// TIA Portal project "IOT2050_S7_CompleteProject" (V16)

(* hardware
DEVICE "ET 200SP station_1"  ET 200SP-Station
   slot 0: "Rack_0"  Rack  6ES5 710-8MAx1
   slot 1: "PLC_1"  CPU 1512SP F-1 PN  6ES7 512-1SK01-0AB0  V2.5
   slot 2: "Server module_1"  Server module  6ES7 193-6PA00-0AA0  V1.1
      slot 1: "Server module_1"  Server module
   slot 127: "BA 2xRJ45"  BA 2xRJ45  6ES7 193-6AR00-0AA0  V0.0
      slot 32769: "Port_1"  6ES7 193-6AR00-0AA0
      slot 32770: "Port_2"  6ES7 193-6AR00-0AA0
*)

// ===== PLC "PLC_1"  CPU 1512SP F-1 PN =====

DATA_BLOCK "motorControl_DB"   // DB2
{ S7_Optimized_Access := 'TRUE' }
VERSION : 0.1
// stored: InstanceOfName motorControl
"motorControl"
BEGIN
END_DATA_BLOCK

// folder: 01_S7

DATA_BLOCK "S7_Data"   // DB1
{ S7_Optimized_Access := 'FALSE' }
VERSION : 0.1
   VAR
      TO_IOT2050 : Struct
         motorCurrent : UInt;   // measured in Amps. Value range (0-255)
         motorVoltage : UInt;   // measured in Volts. Value range (0-255)
         motorTemperature : Real;   // measured in °C
         motorStatus : Bool;   // 0: motor off; 1: motor running (on)
      END_STRUCT;
      FROM_IOT2050 : Struct
         controlButton : Bool;   // button to start or stop motor
      END_STRUCT;
   END_VAR
BEGIN
END_DATA_BLOCK

// folder: (top level)

ORGANIZATION_BLOCK "Main"   // OB1, LAD, ProgramCycle
TITLE = "Main Program Sweep (Cycle)"
{ S7_Optimized_Access := 'TRUE' }
VERSION : 0.1
   VAR_INPUT
      Initial_Call : Bool;   // Initial call of this OB
      Remanence : Bool;   // =True, if remanent data are available
   END_VAR
BEGIN

REGION Network 1
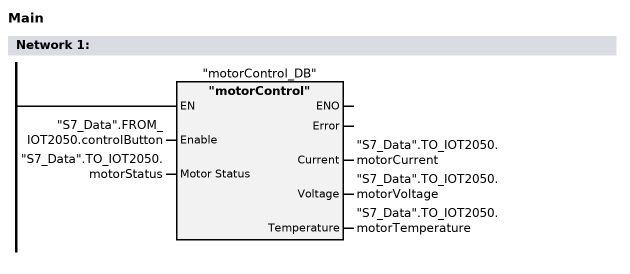
   RUNG wire#powerrail
      "motorControl_DB"(Enable := "S7_Data".FROM_IOT2050.controlButton, "Motor Status" := "S7_Data".TO_IOT2050.motorStatus, Error =>, Current => "S7_Data".TO_IOT2050.motorCurrent, Voltage => "S7_Data".TO_IOT2050.motorVoltage, Temperature => "S7_Data".TO_IOT2050.motorTemperature)
   END_RUNG
   // the same network as SCL:
   "motorControl_DB"(Enable := "S7_Data".FROM_IOT2050.controlButton,   // "motorControl"
                     "Motor Status" := "S7_Data".TO_IOT2050.motorStatus,
                     Current => "S7_Data".TO_IOT2050.motorCurrent,
                     Voltage => "S7_Data".TO_IOT2050.motorVoltage,
                     Temperature => "S7_Data".TO_IOT2050.motorTemperature);
END_REGION
END_ORGANIZATION_BLOCK

// folder: 01_S7

FUNCTION_BLOCK "motorControl"   // FB1, LAD
{ S7_Optimized_Access := 'TRUE' }
VERSION : 0.1
   VAR_INPUT
      Enable : Bool;
   END_VAR
   VAR_OUTPUT
      Error : Bool;
      Current : UInt;
      Voltage : UInt;
      Temperature : Real;
   END_VAR
   VAR_IN_OUT
      "Motor Status" : Bool;
   END_VAR
   VAR
      LGF_SinusCI_Instance : "LGF_SinusCI";
      LGF_RectangleCI_Instance : "LGF_RectangleCI";
   END_VAR
   VAR_TEMP
      randIntError : Bool;
      randIntStatusID : UInt;
      randIntStatus : Word;
      sinusError : Bool;
      sinusStatusID : UInt;
      sinusStatus : Word;
      rectError : Bool;
      rectStatusID : UInt;
      rectStatus : Word;
   END_VAR
BEGIN

REGION Network 1: Set the Motor status to ON/OFF and turn ON/OFF the motor
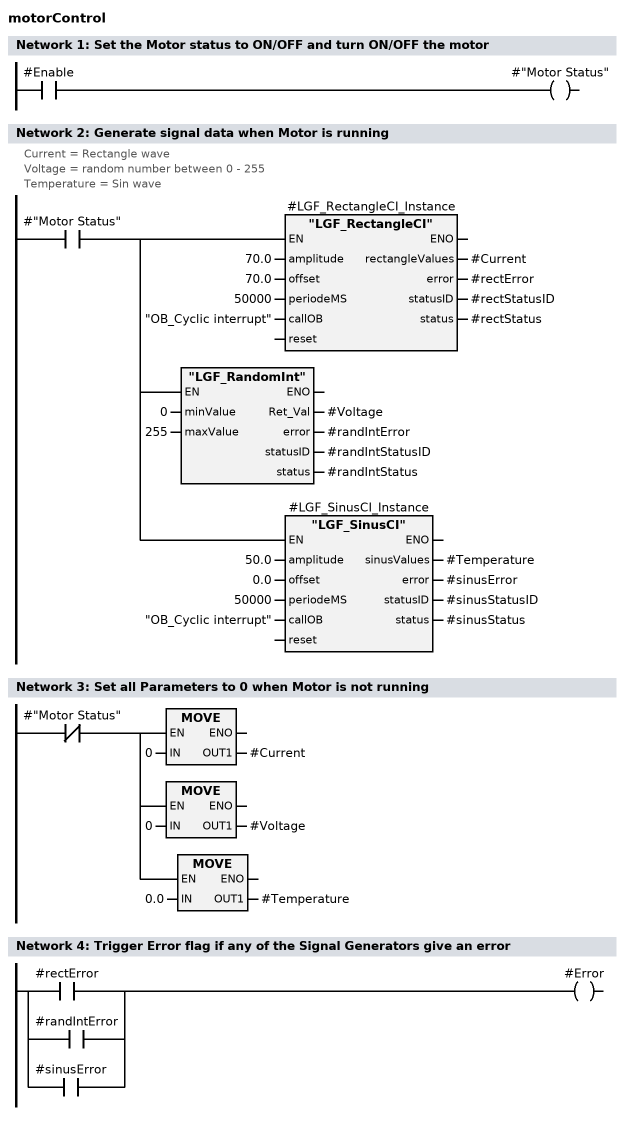
   RUNG wire#powerrail
      Contact( #Enable )
      Coil( #"Motor Status" )
   END_RUNG
   // the same network as SCL:
   #"Motor Status" := #Enable;
END_REGION

REGION Network 2: Generate signal data when Motor is running
   // Current = Rectangle wave
   // Voltage = random number between 0 - 255
   // Temperature = Sin wave
   RUNG wire#powerrail
      Contact( #"Motor Status" )
      wire#w1
      #LGF_RectangleCI_Instance(amplitude := 70.0, offset := 70.0, periodeMS := 50000, callOB := "OB_Cyclic interrupt", reset :=, rectangleValues => #Current, error => #rectError, statusID => #rectStatusID, status => #rectStatus)
   END_RUNG
   RUNG wire#w1
      "LGF_RandomInt"(minValue := 0, maxValue := 255, Ret_Val => #Voltage, error => #randIntError, statusID => #randIntStatusID, status => #randIntStatus)
   END_RUNG
   RUNG wire#w1
      #LGF_SinusCI_Instance(amplitude := 50.0, offset := 0.0, periodeMS := 50000, callOB := "OB_Cyclic interrupt", reset :=, sinusValues => #Temperature, error => #sinusError, statusID => #sinusStatusID, status => #sinusStatus)
   END_RUNG
   // the same network as SCL:
   IF #"Motor Status" THEN
       #LGF_RectangleCI_Instance(amplitude := 70.0,   // "LGF_RectangleCI"
                               offset := 70.0,
                               periodeMS := 50000,
                               callOB := "OB_Cyclic interrupt",
                               rectangleValues => #Current,
                               error => #rectError,
                               statusID => #rectStatusID,
                               status => #rectStatus);
       #Voltage := "LGF_RandomInt"(minValue := 0,
                               maxValue := 255,
                               error => #randIntError,
                               statusID => #randIntStatusID,
                               status => #randIntStatus);
       #LGF_SinusCI_Instance(amplitude := 50.0,   // "LGF_SinusCI"
                             offset := 0.0,
                             periodeMS := 50000,
                             callOB := "OB_Cyclic interrupt",
                             sinusValues => #Temperature,
                             error => #sinusError,
                             statusID => #sinusStatusID,
                             status => #sinusStatus);
   END_IF;
END_REGION

REGION Network 3: Set all Parameters to 0 when Motor is not running
   RUNG wire#powerrail
      I_Contact( #"Motor Status" )
      wire#w1
      Move(in := 0, out1 => #Current)
   END_RUNG
   RUNG wire#w1
      Move(in := 0, out1 => #Voltage)
   END_RUNG
   RUNG wire#w1
      Move(in := 0.0, out1 => #Temperature)
   END_RUNG
   // the same network as SCL:
   IF NOT #"Motor Status" THEN
       #Current := 0;
       #Voltage := 0;
       #Temperature := 0.0;
   END_IF;
END_REGION

REGION Network 4: Trigger Error flag if any of the Signal Generators give an error
   RUNG wire#powerrail
      Contact( #rectError )
      wire#w1
      Coil( #Error )
   END_RUNG
   RUNG wire#powerrail
      Contact( #randIntError )
   END_RUNG wire#w1
   RUNG wire#powerrail
      Contact( #sinusError )
   END_RUNG wire#w1
   // the same network as SCL:
   #Error := #rectError OR #randIntError OR #sinusError;
END_REGION
END_FUNCTION_BLOCK

ORGANIZATION_BLOCK "Cyclic interrupt"   // OB30, LAD, CyclicInterrupt
{ S7_Optimized_Access := 'TRUE' }
VERSION : 0.1
   VAR_INPUT
      Initial_Call : Bool;   // Initial call of this OB
      Event_Count : Int;   // Events discarded
   END_VAR
BEGIN
END_ORGANIZATION_BLOCK

// folder: 01_S7/Signal_Generators

FUNCTION_BLOCK "LGF_SinusCI"   // FB10027, SCL
{ S7_Optimized_Access := 'TRUE' }
VERSION : 0.1
   VAR_INPUT
      amplitude : Real := 0.0;   // Amplitude
      offset : Real := 1000.0;   // Offset
      periodeMS : UDInt := 1000;   // Periode in milliseconds
      callOB : OB_Cyclic;   // Call OB
      reset : Bool;   // Reset values
   END_VAR
   VAR_OUTPUT
      sinusValues : Real;   // Calculated Sinus values
      error : Bool;   // "0" = no error; "1" = error
      statusID : UInt;   // Error source
      status : Word;   // Status and error codes
   END_VAR
   VAR
      statRad : Real;   // Size of an angle in radians
      statCounter : UDInt;   // Counter value
   END_VAR
   VAR_TEMP
      tempCycleTime : UDInt;   // Temp cycle time from CallOB
      tempCyclePhase : UDInt;   // Temp cycle phase from CallOB
      tempCycleStatus : Word;   // Temp cycle status from CallOB
      tempReadTimeStatus : Int;   // Return value of QRY_CINT
   END_VAR
   VAR CONSTANT
      PI : Real := 3.141593;   // PI
      NO_ERROR : Word := 16#0000;   // Status no error
      OB_UNAVAILABLE : Word := 16#8200;   // Status OB not available
      ERROR_IN_THIS_BLOCK : UInt := 1;   // Error ID local error
      ERROR_QRY_CINT : UInt := 2;   // Error ID error in function QRY_CINT
   END_VAR
BEGIN
   //=============================================================================
   // Siemens AG
   // (c)Copyright 2017
   //-----------------------------------------------------------------------------
   // Library:       LGF (Library General Functions)
   // Tested with:   CPU1212C DC/DC/DC FW:V4.2
   // Engineering:   TIA Portal V15 Upd 2
   // Restrictions:  -
   // Requirements:  PLC (S7-1200 / S7-1500)
   // Functionality: This function generates a sinus signal
   //-----------------------------------------------------------------------------
   // Change log table:
   // Version  Date        In charge/Changes applied
   // 01.00.00 03.07.2018  Siemens Industry Online Support
   //                      First released version
   // 01.00.01 17.08.2018  Siemens Industry Online Support
   //                      Upgrade: TIA V15 Update 2
   //-----------------------------------------------------------------------------
   //Status Codes: -
   //=============================================================================

   // Initialize
   #error := FALSE;
   #statusID := #ERROR_IN_THIS_BLOCK;
   #status := #NO_ERROR;

   // get sample time, according to the cyclic interrupt OB number
   #tempReadTimeStatus := QRY_CINT(OB_NR := #callOB, CYCLE => #tempCycleTime,
                                   PHASE => #tempCyclePhase, STATUS => #tempCycleStatus);

   // Generate error message of the QRY_CINT function
   IF (#tempReadTimeStatus <> 0)
   THEN
     #error := TRUE;
     #statusID := #ERROR_QRY_CINT;
     #status := INT_TO_WORD(#tempReadTimeStatus);
     RETURN;
   END_IF;

   // Generate error message when OB unavailable
   IF (#tempCycleStatus = 16#0000)
   THEN
     #error := TRUE;
     #statusID := #ERROR_IN_THIS_BLOCK;
     #status := #OB_UNAVAILABLE;
     RETURN;
   END_IF;

   IF (#reset = TRUE)
   THEN
     #statCounter := 0;
     #sinusValues := 0;
   ELSE
     // Increment Counter with each call of "OB_Cyclic_interrupt"
     #statCounter := #statCounter + (#tempCycleTime) / 1000;
     #statCounter := #statCounter MOD (#periodeMS);

     #statRad := UDINT_TO_REAL(#statCounter) * 2.0 * #PI / (UDINT_TO_REAL(#periodeMS));

     #sinusValues := SIN(#statRad) * #amplitude + #offset;
   END_IF;
END_FUNCTION_BLOCK

FUNCTION_BLOCK "LGF_RectangleCI"   // FB10029, SCL
{ S7_Optimized_Access := 'TRUE' }
VERSION : 0.1
   VAR_INPUT
      amplitude : Real := 0.0;   // Amplitude
      offset : Real := 1000.0;   // Offset
      periodeMS : UDInt := 1000;   // Periode in milliseconds
      callOB : OB_Cyclic;   // Call OB
      reset : Bool;   // Reset values
   END_VAR
   VAR_OUTPUT
      rectangleValues : Real;   // Calculated rectangle values
      error : Bool;   // "0" = no error; "1" = error
      statusID : UInt;   // Error source
      status : Word;   // Status and error codes
   END_VAR
   VAR
      statRad : Real;   // Size of an angle in radians
      statCounter : UDInt;   // Counter value
   END_VAR
   VAR_TEMP
      tempCycleTime : UDInt;   // Temp cycle time from CallOB
      tempCyclePhase : UDInt;   // Temp cycle phase from CallOB
      tempCycleStatus : Word;   // Temp cycle status from CallOB
      tempReadTimeStatus : Int;   // Return value of QRY_CINT
   END_VAR
   VAR CONSTANT
      PI : Real := 3.141593;   // PI
      NO_ERROR : Word := 16#0000;   // Status no error
      OB_UNAVAILABLE : Word := 16#8200;   // Status OB not available
      ERROR_IN_THIS_BLOCK : UInt := 1;   // Error ID local error
      ERROR_QRY_CINT : UInt := 2;   // Error ID error in function QRY_CINT
   END_VAR
BEGIN
   //=============================================================================
   // Siemens AG
   // (c)Copyright 2017
   //-----------------------------------------------------------------------------
   // Library:       LGF (Library General Functions)
   // Tested with:   CPU1212C DC/DC/DC FW:V4.2
   // Engineering:   TIA Portal V15 Upd 2
   // Restrictions:  -
   // Requirements:  PLC (S7-1200 / S7-1500)
   // Functionality: This function generates a rectangle signal
   //-----------------------------------------------------------------------------
   // Change log table:
   // Version  Date        In charge/Changes applied
   // 01.00.00 03.07.2018  Siemens Industry Online Support
   //                      First released version
   // 01.00.01 17.08.2018  Siemens Industry Online Support
   //                      Upgrade: TIA V15 Update 2
   //-----------------------------------------------------------------------------
   //Status Codes: -
   //=============================================================================

   // Initialize
   #error := FALSE;
   #statusID := #ERROR_IN_THIS_BLOCK;
   #status := #NO_ERROR;

   // get sample time, according to the cyclic interrupt OB number
   #tempReadTimeStatus := QRY_CINT(OB_NR := #callOB, CYCLE => #tempCycleTime,
                                   PHASE => #tempCyclePhase, STATUS => #tempCycleStatus);

   // Generate error message of the QRY_CINT function
   IF (#tempReadTimeStatus <> 0)
   THEN
     #error := TRUE;
     #statusID := #ERROR_QRY_CINT;
     #status := INT_TO_WORD(#tempReadTimeStatus);
     RETURN;
   END_IF;

   // Generate error message when OB unavailable
   IF (#tempCycleStatus = 16#0000)
   THEN
     #error := TRUE;
     #statusID := #ERROR_IN_THIS_BLOCK;
     #status := #OB_UNAVAILABLE;
     RETURN;
   END_IF;

   IF (#reset = TRUE) 
   THEN
     #statCounter := 0;
     #rectangleValues := 0;
   ELSE
     // Increment Counter with each call of "OB_Cyclic_interrupt"
     #statCounter := #statCounter + (#tempCycleTime) / 1000;
     #statCounter := #statCounter MOD (#periodeMS);

     IF (#statCounter <= (#periodeMS / 2))
     THEN
       #rectangleValues := #offset + #amplitude;
     ELSE
       #rectangleValues := #offset - #amplitude;
     END_IF;
   END_IF;
END_FUNCTION_BLOCK

FUNCTION "LGF_RandomInt" : Int   // FC10013, SCL
{ S7_Optimized_Access := 'TRUE' }
   VAR_INPUT
      minValue : Int;   // minimal Value random can reach
      maxValue : Int;   // maximal Value random can reach
   END_VAR
   VAR_OUTPUT
      error : Bool;
      statusID : UInt;
      status : Word;
   END_VAR
   VAR_TEMP
      tempTime : DTL;
      tempTimeStatus : Int;
      tempRandomValue : Int;
      tempNormReal : Real;
   END_VAR
   VAR CONSTANT
      NO_ERROR : Word := 16#0000;
      NO_CURRENT_JOBS : Word := 16#7000;
      MAX_LESS_MIN : Word := 16#8200;
      ERROR_IN_THIS_BLOCK : UInt := 1;
      ERROR_RD_SYS_T : UInt := 2;
      MIN_INT : DInt := -32768;
      MAX_INT : DInt := 32767;
   END_VAR
BEGIN
   //=============================================================================
   // Siemens AG
   // (c)Copyright 2017
   //-----------------------------------------------------------------------------
   // Library:       LGF (Library General Functions)
   // Tested with:   CPU1212C DC/DC/DC FW:V4.2
   // Engineering:   TIA Portal V13 SP1 Upd 4
   // Restrictions:  -
   // Requirements:  PLC (S7-1200 / S7-1500)
   // Functionality: This function generates random numbers in defined limits
   //                (Datatype Int)
   //-----------------------------------------------------------------------------
   // Change log table:
   // Version  Date        In charge / Changes applied
   // 01.00.00 19.08.2015  Siemens Industry Online Support
   //                      First released version
   // 01.00.01 02.01.2017  Siemens Industry Online Support
   //                      Upgrade: TIA Portal V14 Update 1
   // 01.00.02 17.08.2018  Siemens Industry Online Support
   //                      Upgrade: TIA V15 Update 2
   //-----------------------------------------------------------------------------
   //Status Codes:
   // 16#7000:  No current jobs
   // 16#0000:  Job finished; Note: There is no "Busy"-Status because the block
   //           is finished within a single cycle
   // 16#8200:  maxValue is samller then minValue 
   //=============================================================================

   //Set "No current job" status
   #error := false;
   #statusID := #ERROR_IN_THIS_BLOCK;
   #status := #NO_CURRENT_JOBS;

   //Check if the maximal Value is less than the minimal value
   IF (#minValue > #maxValue) THEN
     #error := true;
     #statusID := #ERROR_IN_THIS_BLOCK;
     #status := #MAX_LESS_MIN;
     #LGF_RandomInt := 0;
     RETURN;
   END_IF;

   //Read system time
   #tempTimeStatus := RD_SYS_T(#tempTime);

   IF (#tempTimeStatus <> 0) THEN
     #error := true;
     #statusID := #ERROR_RD_SYS_T;
     #status := INT_TO_WORD(#tempTimeStatus);
     #LGF_RandomInt := 0;
     RETURN;
   END_IF;

   //Callculate a random-start-value depending on the time
   #tempRandomValue.%B1 := #tempTime.NANOSECOND.%B0;
   #tempRandomValue.%B0 := #tempTime.NANOSECOND.%B1;

   //adapt the calculated random number to the given number span
   #tempNormReal := NORM_X(MIN := #MIN_INT, VALUE := #tempRandomValue, MAX := #MAX_INT);
   #LGF_RandomInt := SCALE_X(MIN := #minValue, VALUE := #tempNormReal, MAX := #maxValue);

   #status := #NO_ERROR;
END_FUNCTION